// TIA Portal V17 export
// export: Created 2024-09-02T12:50:35.5512314Z, ExportSetting WithDefaults, DisplayName Totally Integrated Automation Portal, DisplayVersion V17, DisplayName TIA Portal Openness, DisplayVersion V17, DisplayName TIA Portal Version Control Interface, DisplayVersion V17, DisplayName STEP 7 Professional, DisplayVersion V17, DisplayName STEP 7 Safety, DisplayVersion V17, DisplayName WinCC Professional, DisplayVersion V17
TYPE "TypeMobyArbeitsPrg_1"
// stored: IsFailsafeCompliant false
   STRUCT
      taf_nr : Int;   // TAF Nummer / TAF number
      taf_vor : Int;   // Taf-Nummer Vorprüfung / Table number Preliminary test
      kennung : Byte;   // Kennung / ID
      arbeitsprg_nr : Byte;   // Arbeitsprogramm / Work program
      takte : Byte;   // Arbeitstakte / Schraubertakte / Working cycles / Screwdriver cycles
      weiterschaltung : Byte;   // TAF-Weiterschaltung 1 - Freigabe, 0 - Automatisch / TAF step-on 1 - Enable, 0 - Automatic
      werkzeug_nr : Int;   // Werkzeugnummer / tool number
      flex_abfrg_byte : Byte;   // Flexible Abfrage Adresse Byte / Flexible query address Byte
      flex_abfrg_bit : Byte;   // Flexible Abfrage Adresse Bit / Flexible query Address Bit
      quell_anbau : Word;   // Quelle Vergleichsdaten / Source Comparative data
      ziel_anbau : Word;   // Ziel der Anbauteile / Aim of the attachments
      meldekntr_1 : Byte;   // Meldekontrollbyte / message control byte
      meldekntr_2 : Byte;   // Meldekontrollbyte / message control byte
      meldekntr_3 : Byte;   // Meldekontrollbyte / message control byte
      meldekntr_4 : Byte;   // Meldekontrollbyte / message control byte
      sonderfunktion : Byte;   // Sonderfunktion / Special functions
      reserve_02 : Byte;   // Reserve
      reserve_03 : Byte;   // Reserve
      reserve_04 : Byte;   // Reserve
   END_STRUCT;
END_TYPE
